(* PLC project real2int_conversion, Dassault Systèmes ControlBuild 2024x *)
(* stored: creationDateTime 2023-10-03T11:13:26-01:00 *)

(* This module converts a real input into an integer output. *)
FUNCTION_BLOCK equipment_library.real2int_conversion
  VAR_INPUT
    input : REAL := 0.0;
  END_VAR
  VAR_OUTPUT
    dintOutput : DINT := 0;
    intOutput : INT := 0;
  END_VAR


ACTION C_source_code:
/* ----------------------------------------------------------------	*/
/* Type : Model of Operative Behaviour					*/
/* Category :  Toolbox							*/
/* Author : Dassault Systemes						*/
/* Update date : June 2018						*/
/* ----------------------------------------------------------------	*/
/* This module converts a real input into an integer ouput.		*/
/* ----------------------------------------------------------------	*/

dintOutput = input;

if ((dintOutput >= -32768) && (dintOutput <= 32767)) 
	intOutput = dintOutput ;
else 
	intOutput = 0;
END_ACTION
END_FUNCTION_BLOCK
